FUNCTION_BLOCK Produce (* Basic Function Block Type *)
  (* Standard: 61499-2 *)
  (* Version 0.0, 9/26/2018, dmidro, nxtControl GmbH, Template *)
  PACKAGE Main;
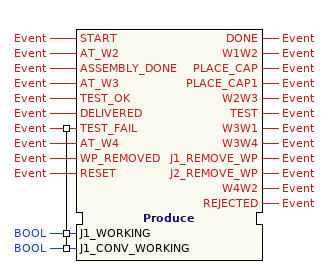
  EVENT_INPUT
    START;
    AT_W2;
    ASSEMBLY_DONE;
    AT_W3;
    TEST_OK;
    DELIVERED;
    TEST_FAIL WITH J1_WORKING, J1_CONV_WORKING;
    AT_W4;
    WP_REMOVED;
    RESET;
  END_EVENT
  EVENT_OUTPUT
    DONE;
    W1W2;
    PLACE_CAP;
    PLACE_CAP1;
    W2W3;
    TEST;
    W3W1;
    W3W4;
    J1_REMOVE_WP;
    J2_REMOVE_WP;
    W4W2;
    REJECTED;
  END_EVENT
  VAR_INPUT
    J1_WORKING : BOOL;
    J1_CONV_WORKING : BOOL;
  END_VAR
  VAR
    PLACE_CAP_VAR : BOOL := TRUE;
  END_VAR
  EC_STATES
    START; (* Initial State *)
    TO_ASSEMBLY : -> W1W2;
    ASSEMBLE : -> PLACE_CAP;
    TO_TEST : -> W2W3;
    TEST : -> TEST;
    TO_OUTPUT : -> W3W1;
    DONE : -> DONE;
    REJECT : -> W3W4;
    REMOVE : -> J1_REMOVE_WP;
    REJECT_DONE : -> REJECTED;
    RESET;
    TO_ASSEMBLY1 : -> W4W2;
    REJECT_J2;
    MOVE_W4 : -> W3W4;
    MOVE_W1 : -> W3W1;
    MOVE_W2_1 : -> W1W2;
    J2_REMOVE : REQ -> J2_REMOVE_WP;
    MOVE_W2_2 : -> W4W2;
    REJECT_DONE2 : -> REJECTED;
    ASSEMBLE1 : -> PLACE_CAP1;
  END_STATES
  EC_TRANSITIONS
    START TO TO_ASSEMBLY := START;
    TO_ASSEMBLY TO ASSEMBLE := AT_W2;
    ASSEMBLE TO TO_TEST := ASSEMBLY_DONE;
    TO_TEST TO TEST := AT_W3;
    TEST TO TO_OUTPUT := TEST_OK;
    TO_OUTPUT TO DONE := DELIVERED;
    DONE TO START := 1;
    TEST TO REJECT := TEST_FAIL AND J1_WORKING;
    REJECT TO REMOVE := AT_W4;
    REMOVE TO REJECT_DONE := WP_REMOVED;
    REJECT_DONE TO TO_ASSEMBLY1 := 1;
    TO_ASSEMBLY TO RESET := RESET;
    ASSEMBLE TO RESET := RESET;
    TO_TEST TO RESET := RESET;
    TEST TO RESET := RESET;
    TO_OUTPUT TO RESET := RESET;
    REJECT TO RESET := RESET;
    REMOVE TO RESET := RESET;
    RESET TO START := 1;
    TO_ASSEMBLY1 TO ASSEMBLE := AT_W2;
    TO_ASSEMBLY1 TO RESET := RESET;
    TEST TO REJECT_J2 := TEST_FAIL AND NOT J1_WORKING;
    REJECT_J2 TO MOVE_W1 := NOT J1_CONV_WORKING;
    REJECT_J2 TO MOVE_W4 := J1_CONV_WORKING;
    MOVE_W4 TO MOVE_W2_2 := AT_W4;
    MOVE_W2_2 TO J2_REMOVE := AT_W2;
    MOVE_W2_1 TO J2_REMOVE := AT_W2;
    MOVE_W1 TO MOVE_W2_1 := DELIVERED;
    J2_REMOVE TO REJECT_DONE2 := WP_REMOVED;
    REJECT_DONE2 TO ASSEMBLE := PLACE_CAP_VAR = TRUE;
    REJECT_DONE2 TO ASSEMBLE1 := PLACE_CAP_VAR = FALSE;
    ASSEMBLE1 TO TO_TEST := ASSEMBLY_DONE;
  END_TRANSITIONS
  ALGORITHM INIT IN ST: (* Initialization algorithm *)
;
  END_ALGORITHM
  ALGORITHM REQ IN ST: (* Normally executed algorithm *)
;
PLACE_CAP_VAR := NOT PLACE_CAP_VAR;
  END_ALGORITHM
END_FUNCTION_BLOCK
